FUNCTION_BLOCK FB_SignalHandling
VAR_INPUT
	bSignalInput			:BOOL;
END_VAR
VAR_OUTPUT
	bSignalOutput			:BOOL;
END_VAR
VAR
	bLocalEnable		:BOOL;
END_VAR

METHOD FB_init : BOOL
VAR_INPUT
	bInitRetains : BOOL; // if TRUE, the retain variables are initialized (warm start / cold start)
	bInCopyCode : BOOL;  // if TRUE, the instance afterwards gets moved into the copy code (online change)	
	
END_VAR
END_METHOD

METHOD SetOutput : BOOL
VAR_INPUT
END_VAR
bSignalOutput := (bLocalEnable AND bSignalInput);
END_METHOD

METHOD SignalEnable : BOOL
VAR_INPUT
	bSignalLocalEnable		:BOOL;
END_VAR
bLocalEnable := bSignalLocalEnable;
END_METHOD

END_FUNCTION_BLOCK

(* stored: Version 1.1.0.1, ProductVersion 3.1.4022.16
   POU FB_SignalHandling: Id {2df786a4-bf08-4249-ad63-77f16f1800cf}, SpecialFunc None
   Method FB_init: Id {41f96695-ff37-483a-9167-37d4dfaa1c92}
   Method SetOutput: Id {61cd6f68-a849-45f6-84dc-71b222c96424}
   Method SignalEnable: Id {b1373d9f-d853-4cdb-9f55-3c60b7fe1632} *)
